{attribute 'linkalways'} 
{attribute 'no_explicit_call' := 'This FB is a CLASS and must be accessed using methods or properties'}
{attribute 'enable_dynamic_creation'}
FUNCTION_BLOCK Node_F_VN_SetImageChannel EXTENDS VisionNode
VAR
    ipSrcImage : _ITcVnImage;
    ipDestImage : _ITcVnImage;
    nSrcChannelIndex : _UINT(0);
    nDestChannelIndex : _UINT(0);
    hrPrev : _HRESULT(S_OK);
	hresult : _HRESULT(S_OK);
END_VAR

METHOD PUBLIC  Clone : I_Node
VAR
	pNode : POINTER TO Node_F_VN_SetImageChannel;
END_VAR
pNode := __NEW(Node_F_VN_SetImageChannel);
Clone := pNode^;
END_METHOD

METHOD FB_init : BOOL
VAR_INPUT
	bInitRetains : BOOL; // if TRUE, the retain variables are initialized (warm start / cold start)
	bInCopyCode : BOOL;  // if TRUE, the instance afterwards gets moved into the copy code (online change)
END_VAR
AddInput('ipSrcImage', ipSrcImage);
AddInput('ipDestImage', ipDestImage);
AddParameter('nSrcChannelIndex', nSrcChannelIndex);
AddParameter('nDestChannelIndex', nDestChannelIndex);
AddInput('hrPrev', hrPrev);
AddOutput('ipDestImage', ipDestImage);
AddOutput('hresult',hresult);
END_METHOD

METHOD PROTECTED OnExecute
hresult.Value := F_VN_SetImageChannel(
    ipSrcImage := ipSrcImage.Value,
	ipDestImage := ipDestImage.Value,
    nSrcChannelIndex := nSrcChannelIndex.Value,
    nDestChannelIndex := nDestChannelIndex.Value,
	hrPrev:= hrPrev.Value);
END_METHOD

METHOD PUBLIC PreExecutionCheck
VAR_INPUT
	Check : I_PreExecutionChecks;
END_VAR
VAR
	srcImageInfo : TcVnImageInfo;
END_VAR
Check.IsTrue(ipSrcImage.IsValid, 'ipSrcImage must contain an image');

IF ipSrcImage.TryGetImageInfo(srcImageInfo) THEN
	Check.IsTrue((nSrcChannelIndex.Value <= srcImageInfo.stPixelFormat.nChannels), 'nSrcChannelIndex is greater than the available ipSrcImage channels');
END_IF

// here
END_METHOD

END_FUNCTION_BLOCK

(* stored: Version 1.1.0.1, ProductVersion 3.1.4024.15
   POU Node_F_VN_SetImageChannel: Id {91eebd60-8725-001c-2ad2-3436ae558f07}, SpecialFunc None
   Folder Constructor: Id {e124acd5-3564-03f3-128b-8c34e13d1977}
   Method Clone: Id {dad9dcfe-97a2-0c90-2958-2145fcc2c334}
   Method FB_init: Id {bb4c9d30-cb67-0977-3850-8cecb5de42d8}
   Method OnExecute: Id {1a467886-dfe5-0839-25c1-b1aab06ab9b8}
   Method PreExecutionCheck: Id {49002dc3-e887-077f-316b-eaebbf25ce5c} *)
